{attribute 'GeneratedUsingTerminal: EPP3752-0000-0017'}
{attribute addProperty BoxType "EPP3752-0000-0017"}
{attribute addProperty Id "EtcSlaveTerminalBaseAI_Inputs_Channel_1AT %I*AI_Inputs_Channel_5A86716D5AI_Inputs_Channel_2AT %I*AI_Inputs_Channel_5A86716D5AI_Inputs_Channel_3AT %I*AI_Inputs_Channel_5A86716D5AI_Inputs_Channel_4AT %I*AI_Inputs_Channel_5A86716D5AI_Inputs_Channel_5AT %I*AI_Inputs_Channel_5A86716D5AI_Inputs_Channel_6AT %I*AI_Inputs_Channel_5A86716D5WcStateAT %I*WcState_9091E0EB2InfoDataAT %I*InfoData_32EB74EA10"}
{attribute addProperty CRC "2488187282"}
{attribute addProperty Size "42"}
TYPE EPP3752_944EB992 EXTENDS EtcSlaveTerminalBase :
STRUCT
	{attribute addProperty Name "AI_Inputs_Channel_1"}
	AI_Inputs_Channel_1 : AI_Inputs_Channel_5A86716D;
	{attribute addProperty Name "AI_Inputs_Channel_2"}
	AI_Inputs_Channel_2 : AI_Inputs_Channel_5A86716D;
	{attribute addProperty Name "AI_Inputs_Channel_3"}
	AI_Inputs_Channel_3 : AI_Inputs_Channel_5A86716D;
	{attribute addProperty Name "AI_Inputs_Channel_4"}
	AI_Inputs_Channel_4 : AI_Inputs_Channel_5A86716D;
	{attribute addProperty Name "AI_Inputs_Channel_5"}
	AI_Inputs_Channel_5 : AI_Inputs_Channel_5A86716D;
	{attribute addProperty Name "AI_Inputs_Channel_6"}
	AI_Inputs_Channel_6 : AI_Inputs_Channel_5A86716D;
	{attribute addProperty Name "WcState"}
	WcState : WcState_9091E0EB;
	{attribute addProperty Name "InfoData"}
	InfoData : InfoData_32EB74EA;
END_STRUCT
END_TYPE

(* stored: Version 1.2.0.0, ProductVersion 3.1.4024.9
   DUT EPP3752_944EB992: Id {db707eb5-3d4e-418b-8d35-acdb6796d987} *)
